TYPE "UDT_WSLStatus"
VERSION : 0.1
   STRUCT
      "010" { ExternalAccessible := 'False'; ExternalVisible := 'False'; ExternalWritable := 'False'} : Struct
         Conveyor { ExternalAccessible := 'False'; ExternalVisible := 'False'; ExternalWritable := 'False'; S7_SetPoint := 'False'} : "UDT_ConveyorStatus";
         PEC_EoS { ExternalAccessible := 'False'; ExternalVisible := 'False'; ExternalWritable := 'False'} : "UDT_PECStatus";
         MCO_M01 { ExternalAccessible := 'False'; ExternalVisible := 'False'; ExternalWritable := 'False'; S7_SetPoint := 'False'} : "UDT_AixControllerStatus";
      END_STRUCT;
      "020" { ExternalAccessible := 'False'; ExternalVisible := 'False'; ExternalWritable := 'False'} : Struct
         Conveyor { ExternalAccessible := 'False'; ExternalVisible := 'False'; ExternalWritable := 'False'; S7_SetPoint := 'False'} : "UDT_ConveyorStatus";
         PEC_EoS { ExternalAccessible := 'False'; ExternalVisible := 'False'; ExternalWritable := 'False'} : "UDT_PECStatus";
         MCO_M01 { ExternalAccessible := 'False'; ExternalVisible := 'False'; ExternalWritable := 'False'; S7_SetPoint := 'False'} : "UDT_AixControllerStatus";
      END_STRUCT;
      "030" { ExternalAccessible := 'False'; ExternalVisible := 'False'; ExternalWritable := 'False'} : Struct
         Conveyor { ExternalAccessible := 'False'; ExternalVisible := 'False'; ExternalWritable := 'False'; S7_SetPoint := 'False'} : "UDT_ConveyorStatus";
         MCO_M01 { ExternalAccessible := 'False'; ExternalVisible := 'False'; ExternalWritable := 'False'; S7_SetPoint := 'False'} : "UDT_AixControllerStatus";
      END_STRUCT;
      "040" { ExternalAccessible := 'False'; ExternalVisible := 'False'; ExternalWritable := 'False'} : Struct
         Conveyor { ExternalAccessible := 'False'; ExternalVisible := 'False'; ExternalWritable := 'False'; S7_SetPoint := 'False'} : "UDT_ConveyorStatus";
         PEC_EoS { ExternalAccessible := 'False'; ExternalVisible := 'False'; ExternalWritable := 'False'} : "UDT_PECStatus";
         MCO_M01 { ExternalAccessible := 'False'; ExternalVisible := 'False'; ExternalWritable := 'False'; S7_SetPoint := 'False'} : "UDT_AixControllerStatus";
      END_STRUCT;
      "050" { ExternalAccessible := 'False'; ExternalVisible := 'False'; ExternalWritable := 'False'} : Struct
         Conveyor { ExternalAccessible := 'False'; ExternalVisible := 'False'; ExternalWritable := 'False'; S7_SetPoint := 'False'} : "UDT_ConveyorStatus";
         PEC_EoS { ExternalAccessible := 'False'; ExternalVisible := 'False'; ExternalWritable := 'False'} : "UDT_PECStatus";
         MCO_M01 { ExternalAccessible := 'False'; ExternalVisible := 'False'; ExternalWritable := 'False'; S7_SetPoint := 'False'} : "UDT_AixControllerStatus";
      END_STRUCT;
      "060" { ExternalAccessible := 'False'; ExternalVisible := 'False'; ExternalWritable := 'False'} : Struct
         Conveyor { ExternalAccessible := 'False'; ExternalVisible := 'False'; ExternalWritable := 'False'; S7_SetPoint := 'False'} : "UDT_ConveyorStatus";
         PEC_EoS { ExternalAccessible := 'False'; ExternalVisible := 'False'; ExternalWritable := 'False'} : "UDT_PECStatus";
         MCO_M01 { ExternalAccessible := 'False'; ExternalVisible := 'False'; ExternalWritable := 'False'; S7_SetPoint := 'False'} : "UDT_AixControllerStatus";
      END_STRUCT;
      "070" { ExternalAccessible := 'False'; ExternalVisible := 'False'; ExternalWritable := 'False'} : Struct
         Conveyor { ExternalAccessible := 'False'; ExternalVisible := 'False'; ExternalWritable := 'False'; S7_SetPoint := 'False'} : "UDT_ConveyorStatus";
         PEC_EoS { ExternalAccessible := 'False'; ExternalVisible := 'False'; ExternalWritable := 'False'} : "UDT_PECStatus";
         MCO_M01 { ExternalAccessible := 'False'; ExternalVisible := 'False'; ExternalWritable := 'False'; S7_SetPoint := 'False'} : "UDT_AixControllerStatus";
      END_STRUCT;
      "080" { ExternalAccessible := 'False'; ExternalVisible := 'False'; ExternalWritable := 'False'} : Struct
         Conveyor { ExternalAccessible := 'False'; ExternalVisible := 'False'; ExternalWritable := 'False'; S7_SetPoint := 'False'} : "UDT_ConveyorStatus";
         PEC_EoS { ExternalAccessible := 'False'; ExternalVisible := 'False'; ExternalWritable := 'False'} : "UDT_PECStatus";
         MCO_M01 { ExternalAccessible := 'False'; ExternalVisible := 'False'; ExternalWritable := 'False'; S7_SetPoint := 'False'} : "UDT_AixControllerStatus";
      END_STRUCT;
      "090" { ExternalAccessible := 'False'; ExternalVisible := 'False'; ExternalWritable := 'False'} : Struct
         Conveyor { ExternalAccessible := 'False'; ExternalVisible := 'False'; ExternalWritable := 'False'; S7_SetPoint := 'False'} : "UDT_ConveyorStatus";
         MCO_M01 { ExternalAccessible := 'False'; ExternalVisible := 'False'; ExternalWritable := 'False'; S7_SetPoint := 'False'} : "UDT_AixControllerStatus";
      END_STRUCT;
      "100" { ExternalAccessible := 'False'; ExternalVisible := 'False'; ExternalWritable := 'False'} : Struct
         Conveyor { ExternalAccessible := 'False'; ExternalVisible := 'False'; ExternalWritable := 'False'; S7_SetPoint := 'False'} : "UDT_ConveyorStatus";
         PEC_EoS { ExternalAccessible := 'False'; ExternalVisible := 'False'; ExternalWritable := 'False'} : "UDT_PECStatus";
         MCO_M01 { ExternalAccessible := 'False'; ExternalVisible := 'False'; ExternalWritable := 'False'; S7_SetPoint := 'False'} : "UDT_AixControllerStatus";
      END_STRUCT;
      "110" { ExternalAccessible := 'False'; ExternalVisible := 'False'; ExternalWritable := 'False'} : Struct
         Conveyor { ExternalAccessible := 'False'; ExternalVisible := 'False'; ExternalWritable := 'False'; S7_SetPoint := 'False'} : "UDT_ConveyorStatus";
         PEC_EoS { ExternalAccessible := 'False'; ExternalVisible := 'False'; ExternalWritable := 'False'} : "UDT_PECStatus";
         MCO_M01 { ExternalAccessible := 'False'; ExternalVisible := 'False'; ExternalWritable := 'False'; S7_SetPoint := 'False'} : "UDT_AixControllerStatus";
      END_STRUCT;
      "120" { ExternalAccessible := 'False'; ExternalVisible := 'False'; ExternalWritable := 'False'} : Struct
         Conveyor { ExternalAccessible := 'False'; ExternalVisible := 'False'; ExternalWritable := 'False'; S7_SetPoint := 'False'} : "UDT_ConveyorStatus";
         MCO_M01 { ExternalAccessible := 'False'; ExternalVisible := 'False'; ExternalWritable := 'False'; S7_SetPoint := 'False'} : "UDT_AixControllerStatus";
      END_STRUCT;
      "121" { ExternalAccessible := 'False'; ExternalVisible := 'False'; ExternalWritable := 'False'} : Struct
         RightAngledTransfer { ExternalAccessible := 'False'; ExternalVisible := 'False'; ExternalWritable := 'False'; S7_SetPoint := 'False'} : "UDT_RATStatus";
         PEC_EoS { ExternalAccessible := 'False'; ExternalVisible := 'False'; ExternalWritable := 'False'; S7_SetPoint := 'False'} : "UDT_PECStatus";
         MCO_M01 { ExternalAccessible := 'False'; ExternalVisible := 'False'; ExternalWritable := 'False'; S7_SetPoint := 'False'} : "UDT_AixControllerStatus";
      END_STRUCT;
      "210" { ExternalAccessible := 'False'; ExternalVisible := 'False'; ExternalWritable := 'False'} : Struct
         Conveyor { ExternalAccessible := 'False'; ExternalVisible := 'False'; ExternalWritable := 'False'; S7_SetPoint := 'False'} : "UDT_ConveyorStatus";
         PEC_EoS { ExternalAccessible := 'False'; ExternalVisible := 'False'; ExternalWritable := 'False'} : "UDT_PECStatus";
         MCO_M01 { ExternalAccessible := 'False'; ExternalVisible := 'False'; ExternalWritable := 'False'; S7_SetPoint := 'False'} : "UDT_AixControllerStatus";
      END_STRUCT;
      "220" { ExternalAccessible := 'False'; ExternalVisible := 'False'; ExternalWritable := 'False'} : Struct
         Conveyor { ExternalAccessible := 'False'; ExternalVisible := 'False'; ExternalWritable := 'False'; S7_SetPoint := 'False'} : "UDT_ConveyorStatus";
         MCO_M01 { ExternalAccessible := 'False'; ExternalVisible := 'False'; ExternalWritable := 'False'; S7_SetPoint := 'False'} : "UDT_AixControllerStatus";
      END_STRUCT;
      "221" { ExternalAccessible := 'False'; ExternalVisible := 'False'; ExternalWritable := 'False'} : Struct
         RightAngledTransfer { ExternalAccessible := 'False'; ExternalVisible := 'False'; ExternalWritable := 'False'; S7_SetPoint := 'False'} : "UDT_RATStatus";
         PEC_EoS { ExternalAccessible := 'False'; ExternalVisible := 'False'; ExternalWritable := 'False'; S7_SetPoint := 'False'} : "UDT_PECStatus";
         MCO_M01 { ExternalAccessible := 'False'; ExternalVisible := 'False'; ExternalWritable := 'False'; S7_SetPoint := 'False'} : "UDT_AixControllerStatus";
      END_STRUCT;
      "230" { ExternalAccessible := 'False'; ExternalVisible := 'False'; ExternalWritable := 'False'} : Struct
         Conveyor { ExternalAccessible := 'False'; ExternalVisible := 'False'; ExternalWritable := 'False'; S7_SetPoint := 'False'} : "UDT_ConveyorStatus";
         MCO_M01 { ExternalAccessible := 'False'; ExternalVisible := 'False'; ExternalWritable := 'False'; S7_SetPoint := 'False'} : "UDT_AixControllerStatus";
      END_STRUCT;
      "240" { ExternalAccessible := 'False'; ExternalVisible := 'False'; ExternalWritable := 'False'} : Struct
         Conveyor { ExternalAccessible := 'False'; ExternalVisible := 'False'; ExternalWritable := 'False'; S7_SetPoint := 'False'} : "UDT_ConveyorStatus";
         PEC_EoS { ExternalAccessible := 'False'; ExternalVisible := 'False'; ExternalWritable := 'False'} : "UDT_PECStatus";
         MCO_M01 { ExternalAccessible := 'False'; ExternalVisible := 'False'; ExternalWritable := 'False'; S7_SetPoint := 'False'} : "UDT_AixControllerStatus";
      END_STRUCT;
      "250" { ExternalAccessible := 'False'; ExternalVisible := 'False'; ExternalWritable := 'False'} : Struct
         Conveyor { ExternalAccessible := 'False'; ExternalVisible := 'False'; ExternalWritable := 'False'; S7_SetPoint := 'False'} : "UDT_ConveyorStatus";
         PEC_EoS { ExternalAccessible := 'False'; ExternalVisible := 'False'; ExternalWritable := 'False'} : "UDT_PECStatus";
         MCO_M01 { ExternalAccessible := 'False'; ExternalVisible := 'False'; ExternalWritable := 'False'; S7_SetPoint := 'False'} : "UDT_AixControllerStatus";
      END_STRUCT;
      "260" { ExternalAccessible := 'False'; ExternalVisible := 'False'; ExternalWritable := 'False'} : Struct
         Conveyor { ExternalAccessible := 'False'; ExternalVisible := 'False'; ExternalWritable := 'False'; S7_SetPoint := 'False'} : "UDT_ConveyorStatus";
         PEC_EoS { ExternalAccessible := 'False'; ExternalVisible := 'False'; ExternalWritable := 'False'} : "UDT_PECStatus";
         MCO_M01 { ExternalAccessible := 'False'; ExternalVisible := 'False'; ExternalWritable := 'False'; S7_SetPoint := 'False'} : "UDT_AixControllerStatus";
      END_STRUCT;
      "270" { ExternalAccessible := 'False'; ExternalVisible := 'False'; ExternalWritable := 'False'} : Struct
         Conveyor { ExternalAccessible := 'False'; ExternalVisible := 'False'; ExternalWritable := 'False'; S7_SetPoint := 'False'} : "UDT_ConveyorStatus";
         MCO_M01 { ExternalAccessible := 'False'; ExternalVisible := 'False'; ExternalWritable := 'False'; S7_SetPoint := 'False'} : "UDT_AixControllerStatus";
      END_STRUCT;
      "280" { ExternalAccessible := 'False'; ExternalVisible := 'False'; ExternalWritable := 'False'} : Struct
         Conveyor { ExternalAccessible := 'False'; ExternalVisible := 'False'; ExternalWritable := 'False'; S7_SetPoint := 'False'} : "UDT_ConveyorStatus";
         PEC_EoS { ExternalAccessible := 'False'; ExternalVisible := 'False'; ExternalWritable := 'False'} : "UDT_PECStatus";
         MCO_M01 { ExternalAccessible := 'False'; ExternalVisible := 'False'; ExternalWritable := 'False'; S7_SetPoint := 'False'} : "UDT_AixControllerStatus";
      END_STRUCT;
      "290" { ExternalAccessible := 'False'; ExternalVisible := 'False'; ExternalWritable := 'False'} : Struct
         Conveyor { ExternalAccessible := 'False'; ExternalVisible := 'False'; ExternalWritable := 'False'; S7_SetPoint := 'False'} : "UDT_ConveyorStatus";
         MCO_M01 { ExternalAccessible := 'False'; ExternalVisible := 'False'; ExternalWritable := 'False'; S7_SetPoint := 'False'} : "UDT_AixControllerStatus";
      END_STRUCT;
      "291" { ExternalAccessible := 'False'; ExternalVisible := 'False'; ExternalWritable := 'False'} : Struct
         RightAngledTransfer { ExternalAccessible := 'False'; ExternalVisible := 'False'; ExternalWritable := 'False'; S7_SetPoint := 'False'} : "UDT_RATStatus";
         PEC_EoS { ExternalAccessible := 'False'; ExternalVisible := 'False'; ExternalWritable := 'False'; S7_SetPoint := 'False'} : "UDT_PECStatus";
         MCO_M01 { ExternalAccessible := 'False'; ExternalVisible := 'False'; ExternalWritable := 'False'; S7_SetPoint := 'False'} : "UDT_AixControllerStatus";
      END_STRUCT;
      "300" { ExternalAccessible := 'False'; ExternalVisible := 'False'; ExternalWritable := 'False'} : Struct
         Conveyor { ExternalAccessible := 'False'; ExternalVisible := 'False'; ExternalWritable := 'False'; S7_SetPoint := 'False'} : "UDT_ConveyorStatus";
         PEC_EoS { ExternalAccessible := 'False'; ExternalVisible := 'False'; ExternalWritable := 'False'} : "UDT_PECStatus";
         MCO_M01 { ExternalAccessible := 'False'; ExternalVisible := 'False'; ExternalWritable := 'False'; S7_SetPoint := 'False'} : "UDT_AixControllerStatus";
      END_STRUCT;
      "410" { ExternalAccessible := 'False'; ExternalVisible := 'False'; ExternalWritable := 'False'} : Struct
         Conveyor { ExternalAccessible := 'False'; ExternalVisible := 'False'; ExternalWritable := 'False'; S7_SetPoint := 'False'} : "UDT_ConveyorStatus";
         PEC_EoS { ExternalAccessible := 'False'; ExternalVisible := 'False'; ExternalWritable := 'False'} : "UDT_PECStatus";
         MCO_M01 { ExternalAccessible := 'False'; ExternalVisible := 'False'; ExternalWritable := 'False'; S7_SetPoint := 'False'} : "UDT_AixControllerStatus";
      END_STRUCT;
      "420" { ExternalAccessible := 'False'; ExternalVisible := 'False'; ExternalWritable := 'False'} : Struct
         Conveyor { ExternalAccessible := 'False'; ExternalVisible := 'False'; ExternalWritable := 'False'; S7_SetPoint := 'False'} : "UDT_ConveyorStatus";
         MCO_M01 { ExternalAccessible := 'False'; ExternalVisible := 'False'; ExternalWritable := 'False'; S7_SetPoint := 'False'} : "UDT_AixControllerStatus";
      END_STRUCT;
      "421" { ExternalAccessible := 'False'; ExternalVisible := 'False'; ExternalWritable := 'False'} : Struct
         RightAngledTransfer { ExternalAccessible := 'False'; ExternalVisible := 'False'; ExternalWritable := 'False'; S7_SetPoint := 'False'} : "UDT_RATStatus";
         PEC_EoS { ExternalAccessible := 'False'; ExternalVisible := 'False'; ExternalWritable := 'False'; S7_SetPoint := 'False'} : "UDT_PECStatus";
         MCO_M01 { ExternalAccessible := 'False'; ExternalVisible := 'False'; ExternalWritable := 'False'; S7_SetPoint := 'False'} : "UDT_AixControllerStatus";
      END_STRUCT;
      "430" { ExternalAccessible := 'False'; ExternalVisible := 'False'; ExternalWritable := 'False'} : Struct
         Conveyor { ExternalAccessible := 'False'; ExternalVisible := 'False'; ExternalWritable := 'False'; S7_SetPoint := 'False'} : "UDT_ConveyorStatus";
         MCO_M01 { ExternalAccessible := 'False'; ExternalVisible := 'False'; ExternalWritable := 'False'; S7_SetPoint := 'False'} : "UDT_AixControllerStatus";
      END_STRUCT;
      "440" { ExternalAccessible := 'False'; ExternalVisible := 'False'; ExternalWritable := 'False'} : Struct
         Conveyor { ExternalAccessible := 'False'; ExternalVisible := 'False'; ExternalWritable := 'False'; S7_SetPoint := 'False'} : "UDT_ConveyorStatus";
         PEC_EoS { ExternalAccessible := 'False'; ExternalVisible := 'False'; ExternalWritable := 'False'} : "UDT_PECStatus";
         MCO_M01 { ExternalAccessible := 'False'; ExternalVisible := 'False'; ExternalWritable := 'False'; S7_SetPoint := 'False'} : "UDT_AixControllerStatus";
      END_STRUCT;
      "450" { ExternalAccessible := 'False'; ExternalVisible := 'False'; ExternalWritable := 'False'} : Struct
         Conveyor { ExternalAccessible := 'False'; ExternalVisible := 'False'; ExternalWritable := 'False'; S7_SetPoint := 'False'} : "UDT_ConveyorStatus";
         PEC_EoS { ExternalAccessible := 'False'; ExternalVisible := 'False'; ExternalWritable := 'False'} : "UDT_PECStatus";
         MCO_M01 { ExternalAccessible := 'False'; ExternalVisible := 'False'; ExternalWritable := 'False'; S7_SetPoint := 'False'} : "UDT_AixControllerStatus";
      END_STRUCT;
      "460" { ExternalAccessible := 'False'; ExternalVisible := 'False'; ExternalWritable := 'False'} : Struct
         Conveyor { ExternalAccessible := 'False'; ExternalVisible := 'False'; ExternalWritable := 'False'; S7_SetPoint := 'False'} : "UDT_ConveyorStatus";
         PEC_EoS { ExternalAccessible := 'False'; ExternalVisible := 'False'; ExternalWritable := 'False'} : "UDT_PECStatus";
         MCO_M01 { ExternalAccessible := 'False'; ExternalVisible := 'False'; ExternalWritable := 'False'; S7_SetPoint := 'False'} : "UDT_AixControllerStatus";
      END_STRUCT;
      "470" { ExternalAccessible := 'False'; ExternalVisible := 'False'; ExternalWritable := 'False'} : Struct
         Conveyor { ExternalAccessible := 'False'; ExternalVisible := 'False'; ExternalWritable := 'False'; S7_SetPoint := 'False'} : "UDT_ConveyorStatus";
         MCO_M01 { ExternalAccessible := 'False'; ExternalVisible := 'False'; ExternalWritable := 'False'; S7_SetPoint := 'False'} : "UDT_AixControllerStatus";
      END_STRUCT;
      "480" { ExternalAccessible := 'False'; ExternalVisible := 'False'; ExternalWritable := 'False'} : Struct
         Conveyor { ExternalAccessible := 'False'; ExternalVisible := 'False'; ExternalWritable := 'False'; S7_SetPoint := 'False'} : "UDT_ConveyorStatus";
         PEC_EoS { ExternalAccessible := 'False'; ExternalVisible := 'False'; ExternalWritable := 'False'} : "UDT_PECStatus";
         MCO_M01 { ExternalAccessible := 'False'; ExternalVisible := 'False'; ExternalWritable := 'False'; S7_SetPoint := 'False'} : "UDT_AixControllerStatus";
      END_STRUCT;
      "490" { ExternalAccessible := 'False'; ExternalVisible := 'False'; ExternalWritable := 'False'} : Struct
         Conveyor { ExternalAccessible := 'False'; ExternalVisible := 'False'; ExternalWritable := 'False'; S7_SetPoint := 'False'} : "UDT_ConveyorStatus";
         MCO_M01 { ExternalAccessible := 'False'; ExternalVisible := 'False'; ExternalWritable := 'False'; S7_SetPoint := 'False'} : "UDT_AixControllerStatus";
      END_STRUCT;
      "491" { ExternalAccessible := 'False'; ExternalVisible := 'False'; ExternalWritable := 'False'} : Struct
         RightAngledTransfer { ExternalAccessible := 'False'; ExternalVisible := 'False'; ExternalWritable := 'False'; S7_SetPoint := 'False'} : "UDT_RATStatus";
         PEC_EoS { ExternalAccessible := 'False'; ExternalVisible := 'False'; ExternalWritable := 'False'; S7_SetPoint := 'False'} : "UDT_PECStatus";
         MCO_M01 { ExternalAccessible := 'False'; ExternalVisible := 'False'; ExternalWritable := 'False'; S7_SetPoint := 'False'} : "UDT_AixControllerStatus";
      END_STRUCT;
      "500" { ExternalAccessible := 'False'; ExternalVisible := 'False'; ExternalWritable := 'False'} : Struct
         Conveyor { ExternalAccessible := 'False'; ExternalVisible := 'False'; ExternalWritable := 'False'; S7_SetPoint := 'False'} : "UDT_ConveyorStatus";
         PEC_EoS { ExternalAccessible := 'False'; ExternalVisible := 'False'; ExternalWritable := 'False'} : "UDT_PECStatus";
         MCO_M01 { ExternalAccessible := 'False'; ExternalVisible := 'False'; ExternalWritable := 'False'; S7_SetPoint := 'False'} : "UDT_AixControllerStatus";
      END_STRUCT;
      "610" { ExternalAccessible := 'False'; ExternalVisible := 'False'; ExternalWritable := 'False'} : Struct
         Conveyor { ExternalAccessible := 'False'; ExternalVisible := 'False'; ExternalWritable := 'False'; S7_SetPoint := 'False'} : "UDT_ConveyorStatus";
         MCO_M01 { ExternalAccessible := 'False'; ExternalVisible := 'False'; ExternalWritable := 'False'; S7_SetPoint := 'False'} : "UDT_AixControllerStatus";
      END_STRUCT;
      "611" { ExternalAccessible := 'False'; ExternalVisible := 'False'; ExternalWritable := 'False'} : Struct
         RightAngledTransfer { ExternalAccessible := 'False'; ExternalVisible := 'False'; ExternalWritable := 'False'; S7_SetPoint := 'False'} : "UDT_RATStatus";
         PEC_EoS { ExternalAccessible := 'False'; ExternalVisible := 'False'; ExternalWritable := 'False'; S7_SetPoint := 'False'} : "UDT_PECStatus";
         MCO_M01 { ExternalAccessible := 'False'; ExternalVisible := 'False'; ExternalWritable := 'False'; S7_SetPoint := 'False'} : "UDT_AixControllerStatus";
      END_STRUCT;
      "620" { ExternalAccessible := 'False'; ExternalVisible := 'False'; ExternalWritable := 'False'} : Struct
         Conveyor { ExternalAccessible := 'False'; ExternalVisible := 'False'; ExternalWritable := 'False'; S7_SetPoint := 'False'} : "UDT_ConveyorStatus";
         MCO_M01 { ExternalAccessible := 'False'; ExternalVisible := 'False'; ExternalWritable := 'False'; S7_SetPoint := 'False'} : "UDT_AixControllerStatus";
      END_STRUCT;
      "630" { ExternalAccessible := 'False'; ExternalVisible := 'False'; ExternalWritable := 'False'} : Struct
         Conveyor { ExternalAccessible := 'False'; ExternalVisible := 'False'; ExternalWritable := 'False'; S7_SetPoint := 'False'} : "UDT_ConveyorStatus";
         MCO_M01 { ExternalAccessible := 'False'; ExternalVisible := 'False'; ExternalWritable := 'False'; S7_SetPoint := 'False'} : "UDT_AixControllerStatus";
      END_STRUCT;
      "640" { ExternalAccessible := 'False'; ExternalVisible := 'False'; ExternalWritable := 'False'} : Struct
         Conveyor { ExternalAccessible := 'False'; ExternalVisible := 'False'; ExternalWritable := 'False'; S7_SetPoint := 'False'} : "UDT_ConveyorStatus";
         PEC_EoS { ExternalAccessible := 'False'; ExternalVisible := 'False'; ExternalWritable := 'False'} : "UDT_PECStatus";
         MCO_M01 { ExternalAccessible := 'False'; ExternalVisible := 'False'; ExternalWritable := 'False'; S7_SetPoint := 'False'} : "UDT_AixControllerStatus";
      END_STRUCT;
   END_STRUCT;

END_TYPE

TYPE "UDT_TGWLiftPI"
VERSION : 0.1
   STRUCT
      ix_SafetyDoorDownDiag : Bool;   // Safety door 1 diagnosis (Lower door)
      ix_MainContactorFeedbackOn : Bool;   // Main Contactor Feedback
      ix_ManualMode : Bool;   // Key-operated switch in manual mode
      ix_AutoMode : Bool;   // Key-operated switch in automatic mode
      ix_JogDown : Bool;   // Push button Jog down
      ix_JogUp : Bool;   // Push button Jog up
      ix_Reset : Bool;   // Push button Reset
      ix_LiftConveyorFwd : Bool;   // Push button lift conveyor foward
      ix_Reference : Bool;   // Pushbutton start lift vertical reference
      ix_InfeedConveyor : Bool;   // Pushbutton infeed conveyor
      ix_LiftConveyorRvs : Bool;   // Push button lift conveyor reverse
      ix_OutfeedConveyor : Bool;   // Pushbutton outfeed conveyor
      ix_SafetyDoorUpDiag : Bool;   // Safety door 1 diagnosis (Upper door)
      Spare_1 : Bool;
      ix_OverTempBrakeRes : Bool;   // Over temperature braking resistor
      Spare_2 : Bool;
      ix_LimSwitchDown : Bool;   // Limit switch down
      ix_LimSwitchUp : Bool;   // Limit switch up
      ix_BeltTearLeft : Bool;   // Belt tear detector left
      ix_BeltTearRight : Bool;   // Belt tear detector right
      ix_MainSwitchCabinetOn : Bool;   // Control panel main switch is on
      ix_F1002ok : Bool;   // Circuit breaker tripped +S1 400 VAC
      ix_F1400ok : Bool;   // Circuit breaker tripped +S1 24 VDC
      ix_MaintenanceSwitchUpOn : Bool;   // Maintenance Switch is on
   END_STRUCT;

END_TYPE

TYPE "UDT_WSLCommonStatus"
VERSION : 0.1
   STRUCT
      "010" { ExternalWritable := 'False'} : "UDT_CommonStatus";
      "020" { ExternalWritable := 'False'} : "UDT_CommonStatus";
      "030" { ExternalWritable := 'False'} : "UDT_CommonStatus";
      "040" { ExternalWritable := 'False'} : "UDT_CommonStatus";
      "050" { ExternalWritable := 'False'} : "UDT_CommonStatus";
      "060" { ExternalWritable := 'False'} : "UDT_CommonStatus";
      "070" { ExternalWritable := 'False'} : "UDT_CommonStatus";
      "080" { ExternalWritable := 'False'} : "UDT_CommonStatus";
      "090" { ExternalWritable := 'False'} : "UDT_CommonStatus";
      "100" { ExternalWritable := 'False'} : "UDT_CommonStatus";
      "110" { ExternalWritable := 'False'} : "UDT_CommonStatus";
      "120" { ExternalWritable := 'False'} : "UDT_CommonStatus";
      "121" { ExternalWritable := 'False'} : "UDT_CommonStatus";
      "210" { ExternalWritable := 'False'} : "UDT_CommonStatus";
      "220" { ExternalWritable := 'False'} : "UDT_CommonStatus";
      "221" { ExternalWritable := 'False'} : "UDT_CommonStatus";
      "230" { ExternalWritable := 'False'} : "UDT_CommonStatus";
      "240" { ExternalWritable := 'False'} : "UDT_CommonStatus";
      "250" { ExternalWritable := 'False'} : "UDT_CommonStatus";
      "260" { ExternalWritable := 'False'} : "UDT_CommonStatus";
      "270" { ExternalWritable := 'False'} : "UDT_CommonStatus";
      "280" { ExternalWritable := 'False'} : "UDT_CommonStatus";
      "290" { ExternalWritable := 'False'} : "UDT_CommonStatus";
      "291" { ExternalWritable := 'False'} : "UDT_CommonStatus";
      "300" { ExternalWritable := 'False'} : "UDT_CommonStatus";
      "410" { ExternalWritable := 'False'} : "UDT_CommonStatus";
      "420" { ExternalWritable := 'False'} : "UDT_CommonStatus";
      "421" { ExternalWritable := 'False'} : "UDT_CommonStatus";
      "430" { ExternalWritable := 'False'} : "UDT_CommonStatus";
      "440" { ExternalWritable := 'False'} : "UDT_CommonStatus";
      "450" { ExternalWritable := 'False'} : "UDT_CommonStatus";
      "460" { ExternalWritable := 'False'} : "UDT_CommonStatus";
      "470" { ExternalWritable := 'False'} : "UDT_CommonStatus";
      "480" { ExternalWritable := 'False'} : "UDT_CommonStatus";
      "490" { ExternalWritable := 'False'} : "UDT_CommonStatus";
      "491" { ExternalWritable := 'False'} : "UDT_CommonStatus";
      "500" { ExternalWritable := 'False'} : "UDT_CommonStatus";
      "610" { ExternalWritable := 'False'} : "UDT_CommonStatus";
      "611" { ExternalWritable := 'False'} : "UDT_CommonStatus";
      "620" { ExternalWritable := 'False'} : "UDT_CommonStatus";
      "630" { ExternalWritable := 'False'} : "UDT_CommonStatus";
      "640" { ExternalWritable := 'False'} : "UDT_CommonStatus";
   END_STRUCT;

END_TYPE

FUNCTION_BLOCK "FB_SickDemoo"
{ S7_Optimized_Access := 'TRUE' }
VERSION : 0.1
   VAR_INPUT
      ix_Trigger { ExternalAccessible := 'False'; ExternalVisible := 'False'; ExternalWritable := 'False'} : Bool;
      HWInputIdent { ExternalAccessible := 'False'; ExternalVisible := 'False'; ExternalWritable := 'False'} : HW_IO := 714;   // Hardware identification number of the input module
      HWInputLength { ExternalAccessible := 'False'; ExternalVisible := 'False'; ExternalWritable := 'False'} : USInt := 32;   // Size of the input module
      HWOutputIdent { ExternalAccessible := 'False'; ExternalVisible := 'False'; ExternalWritable := 'False'} : HW_IO := 716;   // Hardware identification number of the output module
      HWOutputLength { ExternalAccessible := 'False'; ExternalVisible := 'False'; ExternalWritable := 'False'} : USInt := 32;   // Size of the output module
      CANId { ExternalAccessible := 'False'; ExternalVisible := 'False'; ExternalWritable := 'False'} : USInt := 0;   // CAN ID (0= Master / No CAN network)
   END_VAR

   VAR_OUTPUT
      qs_Barcode { ExternalAccessible := 'False'; ExternalVisible := 'False'; ExternalWritable := 'False'} : String;
   END_VAR

   VAR_IN_OUT
      iqUDT_EquipmentControl : "UDT_EquipmentControl";   // Equipment control structure
   END_VAR

   VAR
      IDB_Lector6xx { ExternalAccessible := 'False'; ExternalVisible := 'False'; ExternalWritable := 'False'; S7_SetPoint := 'False'} : "SICK_Lector_CLV6xx_PNDP";
      sa_Inteface { ExternalAccessible := 'False'; ExternalVisible := 'False'; ExternalWritable := 'False'} : Struct
         Outputs { ExternalAccessible := 'False'; ExternalVisible := 'False'; ExternalWritable := 'False'} : Struct
            RdDone { ExternalAccessible := 'False'; ExternalVisible := 'False'; ExternalWritable := 'False'} : Bool;
            ReqDone { ExternalAccessible := 'False'; ExternalVisible := 'False'; ExternalWritable := 'False'} : Bool;
            ReqBusy { ExternalAccessible := 'False'; ExternalVisible := 'False'; ExternalWritable := 'False'} : Bool;
            Error { ExternalAccessible := 'False'; ExternalVisible := 'False'; ExternalWritable := 'False'} : Bool;
            Errorcode { ExternalAccessible := 'False'; ExternalVisible := 'False'; ExternalWritable := 'False'} : DWord;
         END_STRUCT;
         InOut { ExternalAccessible := 'False'; ExternalVisible := 'False'; ExternalWritable := 'False'} : Struct
            Data { ExternalAccessible := 'False'; ExternalVisible := 'False'; ExternalWritable := 'False'; S7_SetPoint := 'False'} : "ST_SICK_Lector_CLV6xx";
         END_STRUCT;
         stEdge { ExternalAccessible := 'False'; ExternalVisible := 'False'; ExternalWritable := 'False'} : Struct   // Edge detection flags
            xEdgeTrigger { ExternalAccessible := 'False'; ExternalVisible := 'False'; ExternalWritable := 'False'} : Bool;
            xEdgeMatchcode { ExternalAccessible := 'False'; ExternalVisible := 'False'; ExternalWritable := 'False'} : Bool;
            xEdgeDone { ExternalAccessible := 'False'; ExternalVisible := 'False'; ExternalWritable := 'False'} : Bool;
            xEdgeError { ExternalAccessible := 'False'; ExternalVisible := 'False'; ExternalWritable := 'False'} : Bool;
            xEdgeTriggerMem { ExternalAccessible := 'False'; ExternalVisible := 'False'; ExternalWritable := 'False'} : Bool;
            xEdgeDoneMem { ExternalAccessible := 'False'; ExternalVisible := 'False'; ExternalWritable := 'False'} : Bool;
            xEdgeErrorMem { ExternalAccessible := 'False'; ExternalVisible := 'False'; ExternalWritable := 'False'} : Bool;
            xEdgeMatchcodeMem { ExternalAccessible := 'False'; ExternalVisible := 'False'; ExternalWritable := 'False'} : Bool;
         END_STRUCT;
         xTrigger { ExternalAccessible := 'False'; ExternalVisible := 'False'; ExternalWritable := 'False'} : Bool;   // Start read tag command
         xMatchcode { ExternalAccessible := 'False'; ExternalVisible := 'False'; ExternalWritable := 'False'} : Bool;
         xTriggerDone { ExternalAccessible := 'False'; ExternalVisible := 'False'; ExternalWritable := 'False'} : Bool;   // Read tag done
         xMatchcodeDone { ExternalAccessible := 'False'; ExternalVisible := 'False'; ExternalWritable := 'False'} : Bool;
         sReadingResult { ExternalAccessible := 'False'; ExternalVisible := 'False'; ExternalWritable := 'False'} : String[200];   // Read content
         stLector { ExternalAccessible := 'False'; ExternalVisible := 'False'; ExternalWritable := 'False'; S7_SetPoint := 'False'} : "ST_SICK_Lector_CLV6xx";   // RFU data
         arrReadingResult { ExternalAccessible := 'False'; ExternalVisible := 'False'; ExternalWritable := 'False'} : Array[0..199] of Byte;   // Read content backup
      END_STRUCT;
      sR_TRIG_Trigger {InstructionName := 'R_TRIG'; LibVersion := '1.0'; ExternalAccessible := 'False'; ExternalVisible := 'False'; ExternalWritable := 'False'; S7_SetPoint := 'False'} : R_TRIG;
      si_GoodRead { ExternalAccessible := 'False'; ExternalVisible := 'False'; ExternalWritable := 'False'} : Int;
      si_No_Read { ExternalAccessible := 'False'; ExternalVisible := 'False'; ExternalWritable := 'False'} : Int;
   END_VAR


BEGIN
	(*----------------------------------------------------------------------------------------
	|                                                                                      |
	|  Function for interacting with Sick  Scanner                                         |
	|                                                                                      |
	|                                                                                      |
	----------------------------------------------------------------------------------------

	Version history:
	Date        | Version   | Author        | Remark
	----------------------------------------------------------------------------------------
	15/11/2023  | 0.1       | S.Nieswiec    | First release
	19/06/2023  | 0.2       | S.Nieswiec    | Changes for BOR site
	25/06/2024  | 0.3       | I.BouAjram    | HW parameters passed from Inputs instead of using hard coding inside the block
	                                        | use of static variables to capture the inputs and outputs of the block
	*)



	#sR_TRIG_Trigger(CLK := #ix_Trigger);

	REGION Scaner Reading & Sorting


	    IF #iqUDT_EquipmentControl.Command.Reset THEN
	        #sa_Inteface.xTriggerDone := FALSE;
	        #sa_Inteface.xTrigger := FALSE;
	    END_IF;

	    IF #sR_TRIG_Trigger.Q THEN
	        #sa_Inteface.xTrigger := TRUE;
	    END_IF;



	    IF #sa_Inteface.xTriggerDone THEN

	        #sa_Inteface.xTrigger := FALSE;
	        #sa_Inteface.xTriggerDone := FALSE;

	        IF #sa_Inteface.sReadingResult[1] = '!' THEN
	            #si_No_Read += 1;
	            #qs_Barcode := 'NoRead';
	        ELSE
	            #si_GoodRead += 1;

	            "FC_ExtractCodeFromString"(is_String := #sa_Inteface.sReadingResult,
	                                       qs_String => #qs_Barcode);

	        END_IF;
	    END_IF;



	END_REGION

	REGION Sick Demo Code
	    (*=========================================================================
	Name: SICK Lector6xx / CLV6xx PROFINET demo
	Author: SICK AG
	===========================================================================
	This demo program enables you open a reading gate using a software trigger
	via the SICK Lector/CLV6xx function block. Furthermore it is possible to
	create a new evaluation condition using the "Matchcode" command.

	The Lector6xx 2D code reader is connected via PROFINET to a Siemens
	S7-1200 PLC.

	Open a reading gate:
	Set the "xTrigger" variable open a reading gate. Please configure the
	device in way, that the reading gate is automatically closed by a
	"good read" condition or after 5 seconds. The "xTriggerDone" flag
	indicates a successful execution of the function and an incoming
	reading result. The "sReadingResult" variable contains the reading
	result (defined in the SOPAS output format) as a string value.

	Matchcode:
	Set the "xMatchcode" variable to create a new matchcode (myMatch) in
	the evaluation conditions of the device. The "xMatchcodeDone" flag
	indicates a successful execution of the function.

	Please use the "Example" watch table to control the program. Use the
	other watch tables to perform further functions of the FB.

	The same example can also been used for a CLV6xx barcode scanner. Please
	configure in this case a CLV6xx instead of a Lector6xx device in
	the hardware configuration of your PLC (GSD settings).
	=========================================================================*)
	(*Function block call*)
	    #IDB_Lector6xx(HWInputIdent := #HWInputIdent,
	                   HWInputLength := #HWInputLength,
	                   HWOutputIdent := #HWOutputIdent,
	                   HWOutputLength := #HWOutputLength,
	                   CANId := #CANId,
	                   TOut := T#10s,
	                   // Req := #sa_Inteface.Inputs.Req,
	                   // TriggerOn := #sa_Inteface.Inputs.TriggerOn,
	                   // TriggerOff := #sa_Inteface.Inputs.TriggerOff,
	                   // Matchcode := #sa_Inteface.Inputs.Matchcode,
	                   // SavePermanent:= #sa_Inteface.Inputs.SavePermanent,
	                   // ComTest := #sa_Inteface.Inputs.ComTest,
	                   // FreeCommand := #sa_Inteface.Inputs.FreeCommand,

	                   Data := #sa_Inteface.InOut.Data,
	                   RdDone => #sa_Inteface.Outputs.RdDone,
	                   ReqDone => #sa_Inteface.Outputs.ReqDone,
	                   ReqBusy => #sa_Inteface.Outputs.ReqBusy,
	                   Error => #sa_Inteface.Outputs.Error,
	                   Errorcode => #sa_Inteface.Outputs.Errorcode


	    );

	(*Edge detection*)
	    #sa_Inteface.stEdge.xEdgeTrigger := #sa_Inteface.xTrigger AND NOT #sa_Inteface.stEdge.xEdgeTriggerMem;
	    #sa_Inteface.stEdge.xEdgeTriggerMem := #sa_Inteface.xTrigger;
	    #sa_Inteface.stEdge.xEdgeMatchcode := #sa_Inteface.xMatchcode AND NOT #sa_Inteface.stEdge.xEdgeMatchcodeMem;
	    #sa_Inteface.stEdge.xEdgeMatchcodeMem := #sa_Inteface.xMatchcode;
	    #sa_Inteface.stEdge.xEdgeDone := #sa_Inteface.Outputs.ReqDone AND NOT #sa_Inteface.stEdge.xEdgeDoneMem;
	    #sa_Inteface.stEdge.xEdgeDoneMem := #IDB_Lector6xx.ReqDone;
	    #sa_Inteface.stEdge.xEdgeError := #IDB_Lector6xx.Error AND NOT #sa_Inteface.stEdge.xEdgeErrorMem;
	    #sa_Inteface.stEdge.xEdgeErrorMem := #sa_Inteface.Outputs.Error;

	(*Function block init: Clear all selection bits*)
	    IF (#sa_Inteface.stEdge.xEdgeTrigger OR #sa_Inteface.stEdge.xEdgeMatchcode) AND NOT #IDB_Lector6xx.ReqBusy THEN
	        //Clear status bits of the example
	        #sa_Inteface.xTriggerDone := FALSE;
	        #sa_Inteface.xMatchcodeDone := FALSE;

	        //Clear selection bits of the function block
	        #IDB_Lector6xx.TriggerOn := FALSE;
	        #IDB_Lector6xx.TriggerOff := FALSE;
	        #IDB_Lector6xx.Matchcode := FALSE;
	        #IDB_Lector6xx.SavePermanent := FALSE;
	        #IDB_Lector6xx.ComTest := FALSE;
	        #IDB_Lector6xx.FreeCommand := FALSE;
	    END_IF;

	(*Start triger device (open the reading gate)*)
	    IF #sa_Inteface.stEdge.xEdgeTrigger AND NOT #IDB_Lector6xx.ReqBusy THEN
	        #IDB_Lector6xx.TriggerOn := TRUE; //Select: Trigger on
	        #IDB_Lector6xx.Req := TRUE; //Start action
	    END_IF;

	(*Start matchcode (creates a new matchcode evaluation condition*)
	    IF #sa_Inteface.stEdge.xEdgeMatchcode AND NOT #IDB_Lector6xx.ReqBusy THEN
	        #sa_Inteface.stLector.Matchcode.sName := 'MyMatch'; //Name of the matchcode condition
	        #sa_Inteface.stLector.Matchcode.nCodeType := '*'; // Code type ('*' = don't care)
	        #sa_Inteface.stLector.Matchcode.iMinMaxLength := 20; //Min and max length code
	        #sa_Inteface.stLector.Matchcode.sContent := 'Sensor Intelligence.'; //Code content

	        #IDB_Lector6xx.Matchcode := TRUE; //Select: Matchcode
	        #IDB_Lector6xx.Req := TRUE; //Start action
	    END_IF;

	(*Incoming reading result*)
	    IF #IDB_Lector6xx.ReqDone THEN
	        IF #sa_Inteface.xTrigger THEN
	            //Copy the data from the reading result structure to a separate array
	            //Only necessary for old S7-1200 controls to parse the data into a string
	            MOVE_BLK(IN := #sa_Inteface.stLector.ReadingResult.arrResult[1],
	                     COUNT := INT_TO_UINT(#sa_Inteface.stLector.ReadingResult.iLength),
	                     OUT => #sa_Inteface.arrReadingResult[0]);

	            // Tranfer the data into a string variable
	            Chars_TO_Strg(Chars := #sa_Inteface.arrReadingResult,
	                          pChars := 0,
	                          Cnt := 0,
	                          Strg => #sa_Inteface.sReadingResult);

	            #sa_Inteface.xTriggerDone := TRUE;
	            #sa_Inteface.xTrigger := FALSE;
	        END_IF;
	    END_IF;

	(*Lector action done*)
	    IF #sa_Inteface.stEdge.xEdgeDone THEN
	        IF #sa_Inteface.xMatchcode THEN
	            #sa_Inteface.xMatchcodeDone := TRUE;
	            #sa_Inteface.xMatchcode := FALSE;
	        END_IF;

	(*Error detected*)
	    ELSIF #sa_Inteface.stEdge.xEdgeError THEN
	        ; //Error handling. The "Errorcode" variable gives your more information about the occured error
	    END_IF;


	    #IDB_Lector6xx.Req := FALSE; //Clear request bit every PLC cycle

	END_REGION
END_FUNCTION_BLOCK

FUNCTION_BLOCK "FB_CountActiveInputs"
{ S7_Optimized_Access := 'TRUE' }
VERSION : 0.1
// ATTRIBUTES
// AUTO_NUMBER = True
// BLOCK_NUMBER = 195
// END_ATTRIBUTES
   VAR_INPUT
      ix_Input1 { ExternalAccessible := 'False'; ExternalVisible := 'False'; ExternalWritable := 'False'} : Bool;   // Bool input 1
      ix_Input2 { ExternalAccessible := 'False'; ExternalVisible := 'False'; ExternalWritable := 'False'} : Bool;   // Bool input 2
      ix_Input3 { ExternalAccessible := 'False'; ExternalVisible := 'False'; ExternalWritable := 'False'} : Bool;   // Bool input 3
      ix_Input4 { ExternalAccessible := 'False'; ExternalVisible := 'False'; ExternalWritable := 'False'} : Bool;   // Bool input 4
      ix_Input5 { ExternalAccessible := 'False'; ExternalVisible := 'False'; ExternalWritable := 'False'} : Bool;   // Bool input 5
      ix_Input6 { ExternalAccessible := 'False'; ExternalVisible := 'False'; ExternalWritable := 'False'} : Bool;   // Bool input 6
      ix_Input7 { ExternalAccessible := 'False'; ExternalVisible := 'False'; ExternalWritable := 'False'} : Bool;   // Bool input 7
      ix_Input8 { ExternalAccessible := 'False'; ExternalVisible := 'False'; ExternalWritable := 'False'} : Bool;   // Bool input 8
      ix_Input9 { ExternalAccessible := 'False'; ExternalVisible := 'False'; ExternalWritable := 'False'} : Bool;   // Bool input 9
      ix_Input10 { ExternalAccessible := 'False'; ExternalVisible := 'False'; ExternalWritable := 'False'} : Bool;   // Bool input 10
      ix_Input11 { ExternalAccessible := 'False'; ExternalVisible := 'False'; ExternalWritable := 'False'} : Bool;   // Bool input 11
      ix_Input12 { ExternalAccessible := 'False'; ExternalVisible := 'False'; ExternalWritable := 'False'} : Bool;   // Bool input 12
      ix_Input13 { ExternalAccessible := 'False'; ExternalVisible := 'False'; ExternalWritable := 'False'} : Bool;   // Bool input 13
      ix_Input14 { ExternalAccessible := 'False'; ExternalVisible := 'False'; ExternalWritable := 'False'} : Bool;   // Bool input 14
      ix_Input15 { ExternalAccessible := 'False'; ExternalVisible := 'False'; ExternalWritable := 'False'} : Bool;   // Bool input 15
      ix_Input16 { ExternalAccessible := 'False'; ExternalVisible := 'False'; ExternalWritable := 'False'} : Bool;   // Bool input 16
   END_VAR

   VAR_OUTPUT
      qi_ActiveInputsCount { ExternalAccessible := 'False'; ExternalVisible := 'False'; ExternalWritable := 'False'} : Int;   // Number of active inputs
   END_VAR

   VAR
      si_I { ExternalAccessible := 'False'; ExternalVisible := 'False'; ExternalWritable := 'False'} : Int;   // FOR Loop index
      sa_BoolArray { ExternalAccessible := 'False'; ExternalVisible := 'False'; ExternalWritable := 'False'} : Array[1..16] of Bool;   // Use an array for the Boolean inputs
   END_VAR


BEGIN
	(*
	----------------------------------------------------------------------------------------

	Version history:
	Date        | Version   | Author        | Remark
	----------------------------------------------------------------------------------------
	22/01/2024  | 1.00      | J.Majer       | Initial version
	12/03/2024  | 1.00      | S. Nieswiec       | Changed ActiveInputsCount to qi_ActiveInputsCount
	*)

	REGION 1 - Initialize counter
	    // On every start of scan initialize output
	    #qi_ActiveInputsCount := 0;

	END_REGION ;
	REGION 2 - Map inputs to array of bool
	    // Map inputs into static array of bools

	    #sa_BoolArray[1] := #ix_Input1;
	    #sa_BoolArray[2] := #ix_Input2;
	    #sa_BoolArray[3] := #ix_Input3;
	    #sa_BoolArray[4] := #ix_Input4;
	    #sa_BoolArray[5] := #ix_Input5;
	    #sa_BoolArray[6] := #ix_Input6;
	    #sa_BoolArray[7] := #ix_Input7;
	    #sa_BoolArray[8] := #ix_Input8;
	    #sa_BoolArray[9] := #ix_Input9;
	    #sa_BoolArray[10] := #ix_Input10;
	    #sa_BoolArray[11] := #ix_Input11;
	    #sa_BoolArray[12] := #ix_Input12;
	    #sa_BoolArray[13] := #ix_Input13;
	    #sa_BoolArray[14] := #ix_Input14;
	    #sa_BoolArray[15] := #ix_Input15;
	    #sa_BoolArray[16] := #ix_Input16;

	END_REGION ;

	REGION 2 - Start active bool counter
	    // with FOR loop search for active bits in array structure and add +1 to output if an input is TRUE

	    FOR #si_I := 1 TO 16 DO
	        IF #sa_BoolArray[#si_I] THEN
	            #qi_ActiveInputsCount := #qi_ActiveInputsCount + 1;
	        END_IF;
	    END_FOR;

	END_REGION ;


END_FUNCTION_BLOCK

FUNCTION_BLOCK "FB_DataLogicBlade"
{ S7_Optimized_Access := 'TRUE' }
VERSION : 0.1
// ATTRIBUTES
// AUTO_NUMBER = True
// BLOCK_NUMBER = 261
// END_ATTRIBUTES
   VAR_INPUT
      iUDT_DataLogic { ExternalAccessible := 'False'; ExternalVisible := 'False'; ExternalWritable := 'False'} : "UDT_DataLogic_IN";   // Data from camera
      ix_trigger { ExternalAccessible := 'False'; ExternalVisible := 'False'; ExternalWritable := 'False'} : Bool;   // Trigger - Activate barcode scanning inside this function
   END_VAR

   VAR_OUTPUT
      qUDT_DataLogic { ExternalAccessible := 'False'; ExternalVisible := 'False'; ExternalWritable := 'False'} : "UDT_DataLogic_OUT";   // Data from PLC to camera
      qs_Barcode { ExternalAccessible := 'False'; ExternalVisible := 'False'; ExternalWritable := 'False'} : String;   // String barcode
      qw_RetVal { ExternalAccessible := 'False'; ExternalVisible := 'False'; ExternalWritable := 'False'} : Word;   // Error code (W#16#...): A - TimeOut; B - Bit from camera "Result available" blocked; C - NO READ; C5 - 5 NO READ in row;  C0 - Empty data from camera; D - Camera Connection Lost; E - incorrect camera config.
   END_VAR

   VAR_IN_OUT
      iqUDT_EquipmentControl : "UDT_EquipmentControl";
   END_VAR

   VAR
      ss_LastResults { ExternalAccessible := 'False'; ExternalVisible := 'False'; ExternalWritable := 'False'} : Struct   // Copy of last result reading barcode value
         DataBarCode { ExternalAccessible := 'False'; ExternalVisible := 'False'; ExternalWritable := 'False'} : Array[0..15] of Char;   // Last barcode
      END_STRUCT;
      ss_Statistic { ExternalAccessible := 'False'; ExternalVisible := 'False'; ExternalWritable := 'False'} : Struct   // All statistics
         st_ActReadingFromCameraTime { ExternalAccessible := 'False'; ExternalVisible := 'False'; ExternalWritable := 'False'} : Time;   // Actual time measurement from trigger to get data from camera
         st_PrevReadingFromCameraTime { ExternalAccessible := 'False'; ExternalVisible := 'False'; ExternalWritable := 'False'} : Time;   // Previous time measurement from trigger to get data from camera
         st_ShortestReadingTime { ExternalAccessible := 'False'; ExternalVisible := 'False'; ExternalWritable := 'False'} : Time;   // The shortest time of reading data from camera  (only OK READ)
         st_LongestReadingTime { ExternalAccessible := 'False'; ExternalVisible := 'False'; ExternalWritable := 'False'} : Time;   // The longest time of reading data from camera  (only OK READ)
         st_AvgReadingTime { ExternalAccessible := 'False'; ExternalVisible := 'False'; ExternalWritable := 'False'} : Time;   // Average time of reading data from camera (only OK READ)
         st_SumOfTimesOkRead { ExternalAccessible := 'False'; ExternalVisible := 'False'; ExternalWritable := 'False'} : Time;   // Sum of all OK READ times - for use in average
         st_ActTimeToNextReady { ExternalAccessible := 'False'; ExternalVisible := 'False'; ExternalWritable := 'False'} : Time;   // Time from trigger to get next high state on bit "Trigger Ready" from camera
         si_OK_READ_CounterGeneral { ExternalAccessible := 'False'; ExternalVisible := 'False'; ExternalWritable := 'False'} : UInt;   // Total number of correct readings
         si_TimeOut_CounterGeneral { ExternalAccessible := 'False'; ExternalVisible := 'False'; ExternalWritable := 'False'} : UInt;   // Total number of timeouts
         si_NO_READ_CounterGeneral { ExternalAccessible := 'False'; ExternalVisible := 'False'; ExternalWritable := 'False'} : UInt;   // Total number of NO READ
         si_NO_READ_CounterInRow { ExternalAccessible := 'False'; ExternalVisible := 'False'; ExternalWritable := 'False'} : UInt;   // Number of No READ in a row (after 5 generate error)
      END_STRUCT;
      ss_prev_Barcode { ExternalAccessible := 'False'; ExternalVisible := 'False'; ExternalWritable := 'False'} : String;   // Previous barcode to compare with the current one to identify a new read
      sdt_TimeStop { ExternalAccessible := 'False'; ExternalVisible := 'False'; ExternalWritable := 'False'} : Date_And_Time;   // Time value read when "phaseOFF"
      sdt_TimeStart { ExternalAccessible := 'False'; ExternalVisible := 'False'; ExternalWritable := 'False'} : Date_And_Time;   // Time value read when trigger occures.
      sdt_TimeOutTime { ExternalAccessible := 'False'; ExternalVisible := 'False'; ExternalWritable := 'False'} : Date_And_Time;   // Constant time measuring for timeout
      st_DiffTimeOutTime { ExternalAccessible := 'False'; ExternalVisible := 'False'; ExternalWritable := 'False'} : Time;   // Time difference: #sdt_TimeOutTime and #sdt_TimeStart.
      st_TimeDiff { ExternalAccessible := 'False'; ExternalVisible := 'False'; ExternalWritable := 'False'} : Time;   // Time defference: #sdt_TimeStop and #sdt_TimeStart
      sw_ErrorCode { ExternalAccessible := 'False'; ExternalVisible := 'False'; ExternalWritable := 'False'} : Word;   // Error code
      s_R_TRIG_Trigger {InstructionName := 'R_TRIG'; LibVersion := '1.0'; ExternalAccessible := 'False'; ExternalVisible := 'False'; ExternalWritable := 'False'; S7_SetPoint := 'False'} : R_TRIG;   // Rising edge trigger signal
      s_R_TRIG_StatisticActCycleTime {InstructionName := 'R_TRIG'; LibVersion := '1.0'; ExternalAccessible := 'False'; ExternalVisible := 'False'; ExternalWritable := 'False'; S7_SetPoint := 'False'} : R_TRIG;   // Rising edge for (#R_TRIG_Result_available.Q OR #sx_ErrorTimeOut)
      s_R_TRIG_NoReadCounter {InstructionName := 'R_TRIG'; LibVersion := '1.0'; ExternalAccessible := 'False'; ExternalVisible := 'False'; ExternalWritable := 'False'; S7_SetPoint := 'False'} : R_TRIG;   // Rising edge for general counter NO_READ
      s_R_TRIG_OkReadCounter {InstructionName := 'R_TRIG'; LibVersion := '1.0'; ExternalAccessible := 'False'; ExternalVisible := 'False'; ExternalWritable := 'False'; S7_SetPoint := 'False'} : R_TRIG;   // Rising edge for general counter OK_READ
      s_R_TRIG_TimeOutCounter {InstructionName := 'R_TRIG'; LibVersion := '1.0'; ExternalAccessible := 'False'; ExternalVisible := 'False'; ExternalWritable := 'False'; S7_SetPoint := 'False'} : R_TRIG;   // Rising edge for general counter TimeOut
      s_R_TRIG_EdgeErrorTimeOut {InstructionName := 'R_TRIG'; LibVersion := '1.0'; ExternalAccessible := 'False'; ExternalVisible := 'False'; ExternalWritable := 'False'; S7_SetPoint := 'False'} : R_TRIG;   // Rising edge for error TimeOut
      s_R_TRIG_ResetStatistics {InstructionName := 'R_TRIG'; LibVersion := '1.0'; ExternalAccessible := 'False'; ExternalVisible := 'False'; ExternalWritable := 'False'; S7_SetPoint := 'False'} : R_TRIG;   // Rising edge for ResetStatistics
      s_R_TRIG_FirstScan {InstructionName := 'R_TRIG'; LibVersion := '1.0'; ExternalAccessible := 'False'; ExternalVisible := 'False'; ExternalWritable := 'False'; S7_SetPoint := 'False'} : R_TRIG;   // Rising edge for mask error TimeOut in first trigger
      s_FB_TimerOnOffDelay_Instance { ExternalAccessible := 'False'; ExternalVisible := 'False'; ExternalWritable := 'False'; S7_SetPoint := 'False'} : "FB_TimerOnOffDelay";
      s_FB_TimerOnOffDelay_Instance_TimeOut_Error { ExternalAccessible := 'False'; ExternalVisible := 'False'; ExternalWritable := 'False'; S7_SetPoint := 'False'} : "FB_TimerOnOffDelay";
      sx_lastResultOK_READ { ExternalAccessible := 'False'; ExternalVisible := 'False'; ExternalWritable := 'False'} : Bool;   // Variable that keeps the OK_READ state of the last scan.
      sx_lastResultNO_READ { ExternalAccessible := 'False'; ExternalVisible := 'False'; ExternalWritable := 'False'} : Bool;   // Variable that keeps the NO_READ state of the last scan.
      sx_BUSY { ExternalAccessible := 'False'; ExternalVisible := 'False'; ExternalWritable := 'False'} : Bool;   // Function is processing data (set with trigger, reset at the end of processing data from the camera)
      sx_InternalTrigger { ExternalAccessible := 'False'; ExternalVisible := 'False'; ExternalWritable := 'False'} : Bool;   // Internal trigger to keep the BladeTrigger active as long as needed.
      sx_PhaseON { ExternalAccessible := 'False'; ExternalVisible := 'False'; ExternalWritable := 'False'} : Bool;   // Signal from the camera given when it is scanning
      sx_PhaseOFF { ExternalAccessible := 'False'; ExternalVisible := 'False'; ExternalWritable := 'False'} : Bool;   // Signal from the camera given when it finishes scanning.
      sx_RecivedData { ExternalAccessible := 'False'; ExternalVisible := 'False'; ExternalWritable := 'False'} : Bool;   // Variable used to store information about the occurrence of "PhaseOFF".
      sx_GeneralFault { ExternalAccessible := 'False'; ExternalVisible := 'False'; ExternalWritable := 'False'} : Bool;   // Any error sets this bit
      sx_ErrorTimeOut { ExternalAccessible := 'False'; ExternalVisible := 'False'; ExternalWritable := 'False'} : Bool;   // Begin measuring time with trigger and finish when camera activate "Results Available". Time set up in constants
      sx_Inter_NO_READ { ExternalAccessible := 'False'; ExternalVisible := 'False'; ExternalWritable := 'False'} : Bool;   // This bit is set when the first character of barcode is '$$'
      sx_Inter_OK_READ { ExternalAccessible := 'False'; ExternalVisible := 'False'; ExternalWritable := 'False'} : Bool;   // This bit is set when the first character of barcode is '!'
      sx_ReceiveNewData { ExternalAccessible := 'False'; ExternalVisible := 'False'; ExternalWritable := 'False'} : Bool;   // This bit is set when the value of the barcode changes (current compared to previous).
      sx_MemoryInterTrig { ExternalAccessible := 'False'; ExternalVisible := 'False'; ExternalWritable := 'False'} : Bool;   // Memory for trigger activation
      sx_FirstTrigger { ExternalAccessible := 'False'; ExternalVisible := 'False'; ExternalWritable := 'False'} : Bool;   // With the first trigger, this bit is set and the program begins to count statistics.
      sx_FirstScan { ExternalAccessible := 'False'; ExternalVisible := 'False'; ExternalWritable := 'False'} : Bool;
      FB_TimerOnOffDelay_Instance { ExternalAccessible := 'False'; ExternalVisible := 'False'; ExternalWritable := 'False'; S7_SetPoint := 'False'} : "FB_TimerOnOffDelay";
   END_VAR

   VAR_TEMP
      ti_TimeCalculation : Int;   // Auxiliary variable for time calculation
   END_VAR

   VAR CONSTANT
      ct_TimeOut : Time := T#20MS;   // TimeOut form Trigger to For camera in DataMan configured 50ms
      ct_PulsTriggerDuration : Time := T#1S;   // Scaning timer. Camera during thise time is scanning and when finish send all codes what read. [ms]
   END_VAR


BEGIN
	(*
	----------------------------------------------------------------------------------------
	|  Stevia Automation Sp.z.o.o                                                          |
	|  Copyright  2024                                                                     |
	|  All Rights Reserved                                                                 |
	                                                                                       |
	----------------------------------------------------------------------------------------

	Version history:
	Date        | Version   | Author             | Remark
	----------------------------------------------------------------------------------------
	23/5/2024   | 0.1       | Grzegorz Czekała    | first release TIA Portal 17 (upd 6)
	24/5/2024   | 0.2       | Grzegorz Czekała    | Change names from Blade200 to "Blade" (this function is universal for both Blade200 and Blade100).
	12/6/2024   | 1.0       | Grzegorz Czekała    | Change the timers, the way the barcode process works. Stop using signals from the camera (OK and NOK).
	                                              | Instead, compare the current barcode with the previous one and check the first character ($$ for OK, ! for NO_READ).
	                                              | Change type of timers on FB_TimerOnOffDelay. Reset all statistic changed from Reset to ResetData in DB_Control
	*)

	REGION 1.0 - Decoding signals from camera and clear temps

	    #sx_PhaseON := #iUDT_DataLogic.DataFromCamera.%X3;
	    #sx_PhaseOFF := #iUDT_DataLogic.DataFromCamera.%X4;

	    #ti_TimeCalculation := 0;

	END_REGION

	REGION 2.0 - Activate trigger PLC output (camera Blade input)

	    #s_R_TRIG_Trigger(CLK := #ix_trigger);  //Rising edge trigger signal
	    #s_R_TRIG_EdgeErrorTimeOut(CLK := #sx_ErrorTimeOut); //Rising edge recive data from camera
	    #s_R_TRIG_FirstScan(CLK := #sx_FirstScan); //Rising edge for mask first scan time out



	    // Activate camera trigger when:, input trigger is activated and previous process is completed
	    IF #s_R_TRIG_Trigger.Q
	        AND NOT #qUDT_DataLogic.BladeTrigger
	        AND NOT #sx_PhaseON
	        AND NOT #sx_PhaseOFF
	        AND NOT #sx_BUSY
	        AND NOT #sx_InternalTrigger
	    THEN
	        #sx_InternalTrigger := TRUE;
	        #sx_BUSY := TRUE;   // process in progress
	        #sx_ErrorTimeOut := FALSE;
	        #sx_RecivedData := FALSE;
	        #sw_ErrorCode := 16#0;
	        #sx_Inter_NO_READ := FALSE;
	        #sx_Inter_OK_READ := FALSE;
	        #sx_FirstTrigger := TRUE;
	    END_IF;

	    REGION 2.1 - Triger duration control

	        IF #sx_InternalTrigger
	        THEN
	            #sx_MemoryInterTrig := true;
	        END_IF;

	        // Control trigger duration
	        #s_FB_TimerOnOffDelay_Instance(iudi_OnDelayTime := TIME_TO_UDINT(#ct_PulsTriggerDuration),
	                                       ix_SignalToDelay := #sx_MemoryInterTrig,
	                                       ix_Enable := TRUE);


	        IF #s_FB_TimerOnOffDelay_Instance.qx_DelayedSignal
	        THEN
	            #sx_MemoryInterTrig := FALSE;

	        END_IF;

	        #qUDT_DataLogic.BladeTrigger := #sx_MemoryInterTrig;


	        // Mask the first time out error, first check result performed value of "ct_TimeOut" before timeout
	        #FB_TimerOnOffDelay_Instance(iudi_OnDelayTime := TIME_TO_UDINT(#ct_PulsTriggerDuration),
	                                     ix_SignalToDelay := #sx_FirstTrigger,
	                                     qx_DelayedSignal => #sx_FirstScan);

	    END_REGION


	END_REGION

	REGION 3.0 - Get data from camera

	    //Important information
	    // Comment for testers: This program can't detect the same barcode twice. When testing, use two or more barcodes alternately.
	    //By default, the camera sends data to the PLC when it finishes calculating.
	    //When connected to DL.CODE software, it calculates immediately, but when it is NOT connected (during normal operation),
	    //it takes about 60 ms to finish calculating after "PhaseOFF".
	    //So, it is important to set up "Send DataOn" /PhaseOFF in DL.CODE. You can find this in "Step2/Good Read Setup -> right side menu".
	    // Camera

	    REGION 3.1 - Copy the last barecode from camera

	        // Copy last result barcode value to DB
	        MOVE_BLK(IN := #iUDT_DataLogic.BarCodeValue[1],
	                 COUNT := 14,
	                 OUT => #ss_LastResults.DataBarCode[1]);

	        IF NOT #sx_FirstTrigger AND NOT #sx_ReceiveNewData
	        THEN
	            FILL_BLK(IN := 1,
	                     COUNT := 14,
	                     OUT => #ss_LastResults.DataBarCode[0]);
	        END_IF;

	        // Conversion from char to string
	        Chars_TO_Strg(Chars := #ss_LastResults.DataBarCode,
	                      pChars := 1,
	                      Cnt := 0,
	                      Strg => #qs_Barcode);


	    END_REGION


	    REGION 3.2 - Control OF NO_READ OR OK_READ sign
	        // When the barcode value changes or a time error occurs, it means a new reading has finished (either successfully or not).
	        IF #sx_FirstTrigger
	            AND (NOT (#ss_prev_Barcode = #qs_Barcode)
	            OR #s_R_TRIG_EdgeErrorTimeOut.Q)
	            OR #s_R_TRIG_FirstScan.Q
	        THEN
	            IF NOT #s_R_TRIG_EdgeErrorTimeOut.Q
	            THEN
	                #sx_ReceiveNewData := true;
	            END_IF;


	            // Copy Last Result NO_READ sign
	            #ss_LastResults.DataBarCode[0] := #iUDT_DataLogic.BarCodeValue0;

	            // Check NO_READ sign
	            IF #ss_LastResults.DataBarCode[0] = '!'
	            THEN
	                #sx_Inter_NO_READ := TRUE;
	                #sx_Inter_OK_READ := FALSE;
	            END_IF;

	            // Check OK_READ sign
	            IF (#ss_LastResults.DataBarCode[0] = '$$')
	                AND NOT #sx_ErrorTimeOut
	            THEN
	                #sx_Inter_OK_READ := TRUE;
	                #sx_Inter_NO_READ := FALSE;
	            END_IF;


	        END_IF;
	    END_REGION

	    REGION 3.3 Storing information OK_READ NO_READ
	        // from the last read FOR analysis purposes
	        IF #sx_ReceiveNewData THEN
	            #sx_lastResultOK_READ := #sx_Inter_OK_READ;
	            #sx_lastResultNO_READ := #sx_Inter_NO_READ;
	        END_IF;
	    END_REGION

	    #ss_prev_Barcode := #qs_Barcode;  // Copy actual value of barecode for the next cycle comparission

	END_REGION

	REGION 4.0 - Statistics

	    REGION 4.1 - Counting OK_READ for calculate averege time

	        // Countup OK_READ

	        #s_R_TRIG_OkReadCounter(CLK := #sx_Inter_OK_READ); //Rising edge of recived OK_READ - has to be here

	        IF #s_R_TRIG_OkReadCounter.Q
	        THEN
	            #ss_Statistic.si_OK_READ_CounterGeneral += 1;
	        END_IF;

	    END_REGION

	    REGION 4.2 - TimeOut error

	        // Copy the start time when the trigger occurs
	        IF #sx_InternalTrigger
	        THEN
	            #ti_TimeCalculation := RD_SYS_T(#sdt_TimeStart);
	        END_IF;

	        // Copy the the end time when the PhaseOff occures
	        IF #sx_ReceiveNewData
	        THEN
	            #sx_RecivedData := TRUE;  // Info that ReceiveNewData
	            #ti_TimeCalculation := RD_SYS_T(#sdt_TimeStop);
	            #st_TimeDiff := T_DIFF(IN1 := #sdt_TimeStop, IN2 := #sdt_TimeStart); // subtracts the times
	        END_IF;

	        //Constant time measuring
	        #ti_TimeCalculation := RD_SYS_T(#sdt_TimeOutTime);
	        #"st_DiffTimeOutTime" := T_DIFF(IN1 := #sdt_TimeOutTime, IN2 := #sdt_TimeStart); // subtracts the times

	        // When the time from trigger to receiving new data is longer than
	        // (trigger duration + ct_TimeOut), it means a Time Out Error has occurred.
	        IF NOT #sx_RecivedData
	            AND (#"st_DiffTimeOutTime"
	            > (#ct_TimeOut + #ct_PulsTriggerDuration))
	        THEN
	            #sx_ErrorTimeOut := TRUE;
	        END_IF;

	        // Counts TimeOut errors
	        IF #s_R_TRIG_EdgeErrorTimeOut.Q
	        THEN
	            #ss_Statistic.si_TimeOut_CounterGeneral += 1;
	        END_IF;


	    END_REGION

	    REGION 4.3 - Time statistics

	        // Time measured from trigger to ReceiveNewData occures
	        #s_R_TRIG_StatisticActCycleTime(CLK := #sx_ReceiveNewData OR #s_R_TRIG_EdgeErrorTimeOut.Q); // This R_Trig have to be here

	        // Sending the time only once in the event of receiving data or exceeding the timeout.
	        IF #s_R_TRIG_StatisticActCycleTime.Q
	        THEN
	            #ss_Statistic.st_PrevReadingFromCameraTime := #ss_Statistic.st_ActReadingFromCameraTime;
	            #ss_Statistic.st_ActReadingFromCameraTime := #st_TimeDiff;

	        END_IF;

	        REGION 4.3.1 - Longest and shortest reading time for OK_READs

	            // Statistics include only OK_READ process
	            IF #sx_Inter_OK_READ AND #sx_ReceiveNewData
	            THEN
	                // Chceck the longest time
	                IF #ss_Statistic.st_ActReadingFromCameraTime > #ss_Statistic.st_LongestReadingTime
	                THEN
	                    #ss_Statistic.st_LongestReadingTime := #ss_Statistic.st_ActReadingFromCameraTime;
	                END_IF;

	                // When PLC startup the shortest time is 0ms, so we put there other start shortest time value
	                IF #ss_Statistic.st_ShortestReadingTime < T#1ms
	                THEN
	                    #ss_Statistic.st_ShortestReadingTime := #ss_Statistic.st_ActReadingFromCameraTime;
	                END_IF;

	                // Chceck the shortest time
	                IF (#ss_Statistic.st_ActReadingFromCameraTime < #ss_Statistic.st_ShortestReadingTime)
	                THEN
	                    #ss_Statistic.st_ShortestReadingTime := #ss_Statistic.st_ActReadingFromCameraTime;
	                END_IF;

	                // Calculate averege Time OF OK_READs
	                #ss_Statistic.st_SumOfTimesOkRead := #ss_Statistic.st_SumOfTimesOkRead + #ss_Statistic.st_ActReadingFromCameraTime;
	                #ss_Statistic.st_AvgReadingTime := #ss_Statistic.st_SumOfTimesOkRead / #ss_Statistic.si_OK_READ_CounterGeneral;

	            END_IF;

	        END_REGION
	    END_REGION

	    REGION 4.4 - Counting NO_READ and NO_READ in a row
	        #s_R_TRIG_NoReadCounter(CLK := #sx_Inter_NO_READ); // This R_Trig has to be here

	        IF #sx_Inter_OK_READ
	        THEN
	            #ss_Statistic.si_NO_READ_CounterInRow := 0;
	        END_IF;


	        IF #s_R_TRIG_NoReadCounter.Q
	        THEN
	            #ss_Statistic.si_NO_READ_CounterGeneral += 1;
	            #ss_Statistic.si_NO_READ_CounterInRow += 1;
	        END_IF;

	    END_REGION
	END_REGION

	REGION 5.0 - THE END - Resets bits AND is READY TO next trigger

	    #sx_InternalTrigger := FALSE;  // Reset on the end first cycle

	    IF #sx_BUSY
	        AND #sx_ReceiveNewData OR #s_R_TRIG_EdgeErrorTimeOut.Q
	    THEN
	        #sx_BUSY := FALSE;

	    END_IF;

	    #sx_ReceiveNewData := FALSE;

	END_REGION

	REGION 6.0 - Reset all statistics

	    // Connects  signals from inputs to reset statistics (either by input bit or input UDT)

	    #s_R_TRIG_ResetStatistics(CLK := #iqUDT_EquipmentControl.Command.ResetData);

	    // Reset all statistic
	    IF #s_R_TRIG_ResetStatistics.Q
	    THEN
	        #ss_Statistic.st_ActReadingFromCameraTime := t#0ms;
	        #ss_Statistic.st_PrevReadingFromCameraTime := t#0ms;
	        #ss_Statistic.st_ShortestReadingTime := t#0ms;
	        #ss_Statistic.st_SumOfTimesOkRead := t#0ms;
	        #ss_Statistic.st_LongestReadingTime := t#0ms;
	        #ss_Statistic.st_ActTimeToNextReady := t#0ms;
	        #ss_Statistic.st_AvgReadingTime := t#0ms;
	        #ss_Statistic.si_OK_READ_CounterGeneral := 0;
	        #ss_Statistic.si_TimeOut_CounterGeneral := 0;
	        #ss_Statistic.si_NO_READ_CounterInRow := 0;
	        #ss_Statistic.si_NO_READ_CounterGeneral := 0;
	        #sx_FirstTrigger := FALSE;
	        #sx_FirstScan := FALSE;
	    END_IF;

	END_REGION

	REGION 7.0 - Errors CODE

	    // Time out
	    IF #sx_ErrorTimeOut
	    THEN
	        #sx_GeneralFault := TRUE;
	        #sw_ErrorCode := 16#800A;
	        #sx_BUSY := FALSE;
	        #sx_PhaseON := FALSE;
	    END_IF;

	    // NO READ
	    IF #sx_Inter_NO_READ
	    THEN
	        #sx_GeneralFault := TRUE;
	        #sw_ErrorCode := 16#800C;     // NO READ
	    END_IF;

	    // 5 NO READ in a row
	    IF #ss_Statistic.si_NO_READ_CounterInRow >= 5
	    THEN
	        #sx_GeneralFault := TRUE;
	        #sw_ErrorCode := 16#805C;    // 5 NO READ in a row
	    END_IF;

	    // Empty data from camera
	    IF (#sx_ReceiveNewData OR #s_R_TRIG_EdgeErrorTimeOut.Q) AND #ss_LastResults.DataBarCode[0] = '$00'
	    THEN
	        #sx_GeneralFault := TRUE;
	        #sw_ErrorCode := 16#80C0;    // Empty data from camera
	    END_IF;

	    // Send error code to output
	    #qw_RetVal := #sw_ErrorCode;

	END_REGION

	REGION 8.0 - Errors reset

	    IF #iqUDT_EquipmentControl.Command.Reset
	    THEN
	        #sx_BUSY := FALSE;
	        #sx_GeneralFault := FALSE;
	        #sw_ErrorCode := 16#0000;
	        #sx_FirstTrigger := FALSE;
	        #sx_FirstScan := FALSE;
	    END_IF;

	END_REGION



END_FUNCTION_BLOCK

TYPE "UDT_TGWLiftConfiguration"
VERSION : 0.1
   STRUCT
      "010" : Struct   // Lift Conveyor configuration
         Conveyor : "UDT_ConveyorConfiguration";   // Conveyor configuration
         PEC_BoS : "UDT_PECConfiguration";   // BoS configuration
         PEC_EoS : "UDT_PECConfiguration";   // EoS configuration
         VFD : "UDT_VfdConfiguration";   // VFD configuration
      END_STRUCT;
      "020" : Struct   // Vertical lift configuration
         VSU : "UDT_VSULiftConfiguration";   // VSU lift configuration
         VFD : "UDT_VfdPositioningConfiguration";   // VFD positioning configuration
      END_STRUCT;
   END_STRUCT;

END_TYPE

TYPE "UDT_Crossoverstatus"
VERSION : 0.1
   STRUCT
      Status { ExternalAccessible := 'False'; ExternalVisible := 'False'; ExternalWritable := 'False'} : Int;   // Common divert status
      Specific { ExternalAccessible := 'False'; ExternalVisible := 'False'; ExternalWritable := 'False'} : Struct
         Up { ExternalAccessible := 'False'; ExternalVisible := 'False'; ExternalWritable := 'False'} : Bool;   // Divert is in Upper position
         Down { ExternalAccessible := 'False'; ExternalVisible := 'False'; ExternalWritable := 'False'} : Bool;   // Divert is in lower position
         Reverse { ExternalAccessible := 'False'; ExternalVisible := 'False'; ExternalWritable := 'False'} : Bool;   // Conveyor is running in reverse direction
         ErrAirpressureNotOk { ExternalAccessible := 'False'; ExternalVisible := 'False'; ExternalWritable := 'False'} : Bool;   // Airpressure is not signalling
         ErrRuntime { ExternalAccessible := 'False'; ExternalVisible := 'False'; ExternalWritable := 'False'} : Bool;   // Divert took too long to move up or down
         ErrOverrun { ExternalAccessible := 'False'; ExternalVisible := 'False'; ExternalWritable := 'False'} : Bool;   // Parcel is in guard PEC, it moved too far and cant be devided
         WarnAirPressure { ExternalAccessible := 'False'; ExternalVisible := 'False'; ExternalWritable := 'False'} : Bool;   // Warning Airpressure is too low
      END_STRUCT;
   END_STRUCT;

END_TYPE

TYPE "UDT_CrossoverConfiguration"
VERSION : 0.1
   STRUCT
      OutfeedTimeOnDelay { ExternalAccessible := 'False'; ExternalVisible := 'False'; ExternalWritable := 'False'} : UDInt;   // PEC on delaytime
      OutfeedTimeOffDelay { ExternalAccessible := 'False'; ExternalVisible := 'False'; ExternalWritable := 'False'} : UDInt;   // PEC off delaytime
      LiftRuntimeUpOnDelay { ExternalAccessible := 'False'; ExternalVisible := 'False'; ExternalWritable := 'False'} : UDInt;   // Runtime delay lifting device up signal on delay
      LiftRuntimeUpOffDelay { ExternalAccessible := 'False'; ExternalVisible := 'False'; ExternalWritable := 'False'} : UDInt;   // Runtime delay lifting device up signal off delay
      LiftRuntimeDownOnDelay { ExternalAccessible := 'False'; ExternalVisible := 'False'; ExternalWritable := 'False'} : UDInt;   // Runtime delay lifting device down signal on delay
      LiftRuntimeDownOffDelay { ExternalAccessible := 'False'; ExternalVisible := 'False'; ExternalWritable := 'False'} : UDInt;   // Runtime delay lifting device down signal off delay
      ParcelDefaultLength { ExternalAccessible := 'False'; ExternalVisible := 'False'; ExternalWritable := 'False'} : Int := 600;   // Default length of parcel
      OutfeedLength { ExternalAccessible := 'False'; ExternalVisible := 'False'; ExternalWritable := 'False'} : Int := 500;   // Length feeding out
      RollerConveyor { ExternalAccessible := 'False'; ExternalVisible := 'False'; ExternalWritable := 'False'} : Struct   // Lower deck settings
         ConveyorLength { ExternalAccessible := 'False'; ExternalVisible := 'False'; ExternalWritable := 'False'} : Int;   // Length of conveyor
         LengthFrom1 { ExternalAccessible := 'False'; ExternalVisible := 'False'; ExternalWritable := 'False'} : Int := 100;   // Offset length to position in [cm] when feeding from conveyor
         LengthFrom2 { ExternalAccessible := 'False'; ExternalVisible := 'False'; ExternalWritable := 'False'} : Int := 100;   // Offset length to position in [cm] when feeding from conveyor
         Runfwd { ExternalAccessible := 'False'; ExternalVisible := 'False'; ExternalWritable := 'False'} : Bool := TRUE;   // When true conveyor is running forward to feed in
      END_STRUCT;
      BeltConveyor { ExternalAccessible := 'False'; ExternalVisible := 'False'; ExternalWritable := 'False'} : Struct   // Upper deck settings
         ConveyorLength { ExternalAccessible := 'False'; ExternalVisible := 'False'; ExternalWritable := 'False'} : Int;   // Length of conveyor
         LengthFrom3 { ExternalAccessible := 'False'; ExternalVisible := 'False'; ExternalWritable := 'False'} : Int := 100;   // Offset length to position in [cm] when feeding from conveyor
         LengthFrom4 { ExternalAccessible := 'False'; ExternalVisible := 'False'; ExternalWritable := 'False'} : Int := 100;   // Offset length to position in [cm] when feeding from conveyor
         Runfwd { ExternalAccessible := 'False'; ExternalVisible := 'False'; ExternalWritable := 'False'} : Bool := TRUE;   // When true conveyor is running forward to feed in
      END_STRUCT;
      Conveyor1 { ExternalAccessible := 'False'; ExternalVisible := 'False'; ExternalWritable := 'False'} : Struct   // Conveyor 1 settings ( set to true is present )
         IsInfeed { ExternalAccessible := 'False'; ExternalVisible := 'False'; ExternalWritable := 'False'} : Bool := TRUE;   // Is upstream conveyor
         IsOutfeed { ExternalAccessible := 'False'; ExternalVisible := 'False'; ExternalWritable := 'False'} : Bool;   // Is downstream conveyor
      END_STRUCT;
      Conveyor2 { ExternalAccessible := 'False'; ExternalVisible := 'False'; ExternalWritable := 'False'} : Struct   // Conveyor 2 settings ( set to true is present )
         IsInfeed { ExternalAccessible := 'False'; ExternalVisible := 'False'; ExternalWritable := 'False'} : Bool;   // Is upstream conveyor
         IsOutfeed { ExternalAccessible := 'False'; ExternalVisible := 'False'; ExternalWritable := 'False'} : Bool := TRUE;   // Is downstream conveyor
      END_STRUCT;
      Conveyor3 { ExternalAccessible := 'False'; ExternalVisible := 'False'; ExternalWritable := 'False'} : Struct   // Conveyor 3 settings ( set to true is present )
         IsInfeed { ExternalAccessible := 'False'; ExternalVisible := 'False'; ExternalWritable := 'False'} : Bool := TRUE;   // Is upstream conveyor
         IsOutfeed { ExternalAccessible := 'False'; ExternalVisible := 'False'; ExternalWritable := 'False'} : Bool;   // Is downstream conveyor
      END_STRUCT;
      Conveyor4 { ExternalAccessible := 'False'; ExternalVisible := 'False'; ExternalWritable := 'False'} : Struct   // Conveyor 4 settings ( set to true is present )
         IsInfeed { ExternalAccessible := 'False'; ExternalVisible := 'False'; ExternalWritable := 'False'} : Bool := TRUE;   // Is upstream conveyor
         IsOutfeed { ExternalAccessible := 'False'; ExternalVisible := 'False'; ExternalWritable := 'False'} : Bool;   // Is downstream conveyor
      END_STRUCT;
   END_STRUCT;

END_TYPE

FUNCTION "FC_HMDecodeHeader" : Void
{ S7_Optimized_Access := 'TRUE' }
VERSION : 0.1
// ATTRIBUTES
// AUTO_NUMBER = True
// BLOCK_NUMBER = 41
// END_ATTRIBUTES
   VAR_INPUT
      iUDT_FifoMsg : "UDT_Message";   // Buffer for FIFO's message
   END_VAR

   VAR_OUTPUT
      qUDT_MSG : "UDT_HMMessageHeader";   // Messade header structure
   END_VAR

   VAR_TEMP
      ts_MessageHeader : String[15];
      ti_SizeOfMsg : Int;
      ti_Position : Int;
   END_VAR

   VAR CONSTANT
      cc_DL : Char := '$1D';   // Comma sign
   END_VAR


BEGIN
	(*
	----------------------------------------------------------------------------------------

	Version history:
	Date        | Version   | Author        | Remark
	----------------------------------------------------------------------------------------
	27/10/2021  | 0.1       | J.Krawczuk    | first release MHS TIA 15.1
	18/11/2021  | 0.2       | M.Piela       | Interface changes
	*)

	REGION - 1 Header decode


	    #qUDT_MSG.STX := #iUDT_FifoMsg.Character[0];

	    Chars_TO_Strg(Chars := #iUDT_FifoMsg.Character,
	                  pChars := 1,
	                  Cnt := 4,
	                  Strg => #qUDT_MSG.PLCID);

	    Chars_TO_Strg(Chars := #iUDT_FifoMsg.Character,
	                  pChars := 6,
	                  Cnt := 8,
	                  Strg => #qUDT_MSG.SequenceNumber);

	    Chars_TO_Strg(Chars := #iUDT_FifoMsg.Character,
	                  pChars := 15,
	                  Cnt := 15,
	                  Strg => #ts_MessageHeader);

	    #ti_Position := FIND(IN1 := #ts_MessageHeader, IN2 := #cc_DL);

	    Chars_TO_Strg(Chars := #iUDT_FifoMsg.Character,
	                  pChars := 15,
	                  Cnt := INT_TO_UINT(#ti_Position - 1),
	                  Strg => #qUDT_MSG.MessageHeader);

	END_REGION



END_FUNCTION

TYPE "UDT_PushUpDivertCommand"
VERSION : 0.1
   STRUCT
      ManualStartStop : Bool;   // Run conveyor in manual mode
      ManualFullSpeed : Bool;   // Full speed conveyor in manual mode
      ManualJog : Bool;   // Command to jog conveyor in slow speed from HMI
      Reverse : Bool;   // Command to run conveyor in reverse direction from HMI
      ManualSpeed : Int := 50;   // Manual mode speed as percentage of nominal speed [0-100%]
      ManualMode : Bool;   // Manual mode command from HMI
      ManualUp : Bool;   // Command to move devise up
      ManualDown : Bool;   // Command to move devise down
   END_STRUCT;

END_TYPE

TYPE "UDT_PushUpDivertStatus"
VERSION : 0.1
   STRUCT
      Status { ExternalAccessible := 'False'; ExternalVisible := 'False'; ExternalWritable := 'False'} : Int;   // Common divert status
      Specific { ExternalAccessible := 'False'; ExternalVisible := 'False'; ExternalWritable := 'False'} : Struct
         Up { ExternalAccessible := 'False'; ExternalVisible := 'False'; ExternalWritable := 'False'} : Bool;   // Divert is in Upper position
         Down { ExternalAccessible := 'False'; ExternalVisible := 'False'; ExternalWritable := 'False'} : Bool;   // Divert is in lower position
         Reverse { ExternalAccessible := 'False'; ExternalVisible := 'False'; ExternalWritable := 'False'} : Bool;   // Conveyor is running in reverse direction
         ErrAirpressureNotOk { ExternalAccessible := 'False'; ExternalVisible := 'False'; ExternalWritable := 'False'} : Bool;   // Airpressure is not signalling
         ErrRuntime { ExternalAccessible := 'False'; ExternalVisible := 'False'; ExternalWritable := 'False'} : Bool;   // Divert took too long to move up or down
         ErrOverrun { ExternalAccessible := 'False'; ExternalVisible := 'False'; ExternalWritable := 'False'} : Bool;   // Parcel is in guard PEC, it moved too far and cant be devided
         WarnAirPressure { ExternalAccessible := 'False'; ExternalVisible := 'False'; ExternalWritable := 'False'} : Bool;   // Warning Airpressure is too low
      END_STRUCT;
   END_STRUCT;

END_TYPE

TYPE "UDT_PushUpDivertConfiguration"
VERSION : 0.1
   STRUCT
      PECTriggerTimeOnDelay { ExternalAccessible := 'False'; ExternalVisible := 'False'; ExternalWritable := 'False'; S7_SetPoint := 'True'} : UDInt;   // Time after which PEC full is detected
      PECTriggerTimeOffDelay { ExternalAccessible := 'False'; ExternalVisible := 'False'; ExternalWritable := 'False'; S7_SetPoint := 'True'} : UDInt;   // Time after which PEC full is released
      PECLeftTimeOnDelay { ExternalAccessible := 'False'; ExternalVisible := 'False'; ExternalWritable := 'False'; S7_SetPoint := 'True'} : UDInt;   // Time after which PEC full is detected
      PECLeftTimeOffDelay { ExternalAccessible := 'False'; ExternalVisible := 'False'; ExternalWritable := 'False'; S7_SetPoint := 'True'} : UDInt;   // Time after which PEC full is released
      PECRightTimeOnDelay { ExternalAccessible := 'False'; ExternalVisible := 'False'; ExternalWritable := 'False'; S7_SetPoint := 'True'} : UDInt;   // Time after which PEC full is detected
      PECRightTimeOffDelay { ExternalAccessible := 'False'; ExternalVisible := 'False'; ExternalWritable := 'False'; S7_SetPoint := 'True'} : UDInt;   // Time after which PEC full is released
      DivertMonitorUpOnDelay { ExternalAccessible := 'False'; ExternalVisible := 'False'; ExternalWritable := 'False'; S7_SetPoint := 'True'} : UDInt := 1000;   // Time after which sensor up is detected
      DivertMonitorUPOffDelay { ExternalAccessible := 'False'; ExternalVisible := 'False'; ExternalWritable := 'False'; S7_SetPoint := 'True'} : UDInt;   // Time after which sensor up is released
      DivertMonitorDownOnDelay { ExternalAccessible := 'False'; ExternalVisible := 'False'; ExternalWritable := 'False'; S7_SetPoint := 'True'} : UDInt := 1000;   // Time after which sensor down is detected
      DivertMonitorDownOffDelay { ExternalAccessible := 'False'; ExternalVisible := 'False'; ExternalWritable := 'False'; S7_SetPoint := 'True'} : UDInt;   // Time after which sensor down is released
      "Conveyor length" { ExternalAccessible := 'False'; ExternalVisible := 'False'; ExternalWritable := 'False'; S7_SetPoint := 'True'} : Int := 1000;   // Length of the conveyor [mm]
      DecisionPoint { ExternalAccessible := 'False'; ExternalVisible := 'False'; ExternalWritable := 'False'; S7_SetPoint := 'True'} : Int := 1000;   // Point of decision [mm]
      ParcelDefaultLength { ExternalAccessible := 'False'; ExternalVisible := 'False'; ExternalWritable := 'False'; S7_SetPoint := 'True'} : Int := 600;   // Default length of the parcel if none was measured in [mm]
      LengthIn { ExternalAccessible := 'False'; ExternalVisible := 'False'; ExternalWritable := 'False'; S7_SetPoint := 'True'} : Int := 450;   // Length travelling in [mm]
      LengthOut { ExternalAccessible := 'False'; ExternalVisible := 'False'; ExternalWritable := 'False'; S7_SetPoint := 'True'} : Int := 450;   // Length travelling out [mm]
      PositionOffset { ExternalAccessible := 'False'; ExternalVisible := 'False'; ExternalWritable := 'False'; S7_SetPoint := 'True'} : Int;   // Offset to position parcel to compensate speed and weight
      SizeDivert { ExternalAccessible := 'False'; ExternalVisible := 'False'; ExternalWritable := 'False'; S7_SetPoint := 'True'} : Bool := TRUE;   // When true divert is done based on dimension of parcel
   END_STRUCT;

END_TYPE

TYPE "UDT_NerakLiftStatistics"
VERSION : 0.1
   STRUCT
      ProductFellDown : "UDT_EventStatistic";
      CollisionDetected : "UDT_EventStatistic";
      EnergySave : "UDT_EventStatistic";   // Number of times that save energy mode occurs
      ConveyorUp : "UDT_EventStatistic";   // Conveyor up statistics
      ConveyorDown : "UDT_EventStatistic";   // Conveyor down statistics
      ConveyorStop : "UDT_EventStatistic";   // Conveyor down statistics
   END_STRUCT;

END_TYPE

